FUNCTION_BLOCK FB_NormalWash IMPLEMENTS I_WashStrategy
VAR
	   stWashSettings   : ST_WashSettings;
     bStarted   : BOOL := FALSE;
END_VAR

METHOD FB_init : BOOL
VAR_INPUT
	bInitRetains : BOOL; // if TRUE, the retain variables are initialized (warm start / cold start)
	bInCopyCode : BOOL;  // if TRUE, the instance afterwards gets moved into the copy code (online change)
END_VAR
stWashSettings.tFillDuration  := GVL_WashConstants.NORMAL_FILL;
stWashSettings.tWashDuration  := GVL_WashConstants.NORMAL_WASH;
stWashSettings.tDrainDuration := GVL_WashConstants.NORMAL_DRAIN;
stWashSettings.rWashTemperature   := GVL_WashConstants.NORMAL_TEMP;
stWashSettings.nSpinSpeed     := GVL_WashConstants.NORMAL_SPEED;
stWashSettings.sDescription   := 'Soft wash — gentle cycle low temp';

FB_init := TRUE;
END_METHOD

{warning 'add method implementation '}
METHOD GetDuration : TIME
GetDuration := stWashSettings.tWashDuration;
END_METHOD

{warning 'add method implementation '}
METHOD GetProgramName : STRING
GetProgramName := 'NORMAL WASH';
END_METHOD

{warning 'add method implementation '}
METHOD GetWashSettings : ST_WashSettings
GetWashSettings := stWashSettings;
END_METHOD

{warning 'add method implementation '}
METHOD Start : BOOL
bStarted := TRUE;
Start     := TRUE;
END_METHOD

END_FUNCTION_BLOCK

(* stored: Version 1.1.0.1, ProductVersion 3.1.4024.16
   POU FB_NormalWash: Id {298539ff-2152-4423-93cb-375cb98e3ef0}, SpecialFunc None
   Method FB_init: Id {5aaa6437-4752-4a14-b198-2725c5f9c4b8}
   Method GetDuration: Id {fe08b972-8461-481c-acc5-2a5693623f1c}
   Method GetProgramName: Id {0fc7225e-8b67-4de1-9e13-6065c77f91e6}
   Method GetWashSettings: Id {a80a829e-cfac-4213-9b0d-2547a850b7c6}
   Method Start: Id {958a902d-b70e-4272-b36d-0dd8cdb4ab55} *)
